(* CODESYS project FRAME_TWB.visu.xml

Project tree, tasks and I/O mapping:
  visualisation FRAME_TWB
*)

// /FRAME_TWB
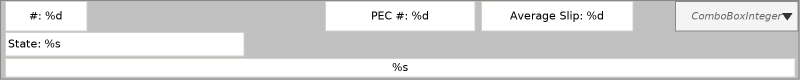
VISUALIZATION FRAME_TWB  // 800x80
VAR_IN_OUT
	conveyor : DUT_CONV_FRAME;
END_VAR
    Textfield (5,58 790x19), "%s", text variable: conveyor.asciiString
    ComboBoxInteger (675,1 123x30), variable: conveyor.dimension, text list: 'TextList_dimensions'
    Textfield (5,1 82x30), "#: %d", text variable: conveyor.conv_number
        OnMouseClick: write the text variable via Default, min 0, max 4
    Textfield (325,1 150x30), "PEC #: %d", text variable: conveyor.pec_idx
        OnMouseClick: write the text variable via Default, min 1, max 10
    Textfield (481,1 152x30), "Average Slip: %d", text variable: conveyor.pecAverageSlip
    Textfield (5,32 239x24), "State: %s", text variable: conveyor.state
END_VISUALIZATION
